PROGRAM AppliedMathematics

END_PROGRAM

(* stored: Version 1.1.0.1
   POU AppliedMathematics: Id {eae2ffb1-ad5a-46f8-8346-f2d4784b446a}, SpecialFunc None *)
